// TwinCAT 3 PLC project PLC
// ProgramVersion: 3.1.4026.19
// CompilerDefines: VISU_USEPROPERTYINFO
// libraries:
//   Tc2_Standard, * (Beckhoff Automation GmbH)
//   Tc2_System, * (Beckhoff Automation GmbH)
// project tree:
//   / GlobalTextList.TcGTLO, PlcTask.TcTTO, Visualization Manager.TcVMO (not stored)
//   POUs/ MAIN.TcPOU
//   VISUs/ Visualization.TcVIS
// real-time tasks:
//   TASK PlcTask: cycle T#10ms, priority 20, ADS port 350
// I/O:
//   DEVICE Device 1 (EtherCAT), AmsNetId 192.168.91.1.2.1
//     Term 1 (EK1100) [EK1100 EtherCAT Coupler (2A E-Bus)]
//       Term 2 (EL2004) [EL2004 4Ch. Dig. Output 24V, 0.5A]
//       Term 3 (EL1004) [EL1004 4Ch. Dig. Input 24V, 3ms]
// variable links:
//   PLC/PLC Instance <-> Device 1 (EtherCAT)/Term 1 (EK1100)/Term 2 (EL2004)
//     PlcTask Outputs/MAIN.bMainMotor <-> Channel 1/Output
//   PLC/PLC Instance <-> Device 1 (EtherCAT)/Term 1 (EK1100)/Term 3 (EL1004)
//     PlcTask Inputs/MAIN.bHardwareButton <-> Channel 1/Input

CONFIGURATION PLC
    RESOURCE PLC ON TwinCAT3
        TASK PlcTask(INTERVAL := T#10ms, PRIORITY := 20);
        PROGRAM MAIN WITH PlcTask : MAIN;
    END_RESOURCE
END_CONFIGURATION

// ---- POUs/MAIN.TcPOU
PROGRAM MAIN
VAR
	
	bHardwareButton AT %I* : BOOL;
	
	bHmiButton : BOOL;
	
	bMainMotor AT %Q* : BOOL;
	
END_VAR

bMainMotor := bHardwareButton or bHmiButton;

END_PROGRAM

// ---- VISUs/Visualization.TcVIS
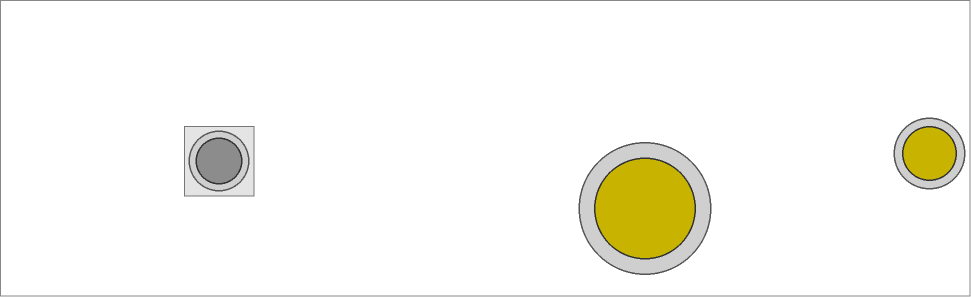
VISUALIZATION Visualization  // 971x297
    PushSwitch (184,126 70x70), variable: MAIN.bHmiButton, behaviour: TOGGLE, style: Switch-PushSwitch-Gray
    Lamp1 (568,120 154x177), variable: MAIN.bMainMotor, style: Lamp-Lamp1-Yellow
    Lamp1 (888,111 83x85), variable: MAIN.bHardwareButton, style: Lamp-Lamp1-Yellow
END_VISUALIZATION
